// Mitsubishi GX Works2 project: PLC_GROUP_37   PLC: FX3G

// global labels: Global1
VAR_GLOBAL
  Day_Active_Light AT Y007 : BOOL;
  Emergency_Stop AT X005 : BOOL;
  Start_Day_Switch AT X007 : BOOL;
  Raspberry_Stock AT D1110 : REAL;
  Lemon_Stock AT D1120 : REAL;
  Stabilizer_Stock AT D1130 : REAL;
  Gummy_Stock AT D1140 : REAL;
  Total_Packages AT D1150 : REAL;
  Raspberry_Input AT D1160 : REAL;
  Lemon_Input AT D1170 : REAL;
  Stabilizer_Input AT D1180 : REAL;
  Gummy_Input AT D1190 : REAL;
END_VAR
VAR_GLOBAL CONSTANT
  Constant_0 : REAL;
END_VAR
VAR_GLOBAL
  End_Day_Flag AT M0 : BOOL;
  Start_Production_Switch AT X001 : BOOL;
  Analog_Input_1 AT D8280 : INT;
  Sampled_Package_Type AT D1100 : REAL;
  Regular_Selected AT M1 : BOOL;
  Luxury_Selected AT M3 : BOOL;
  Inventory_OK AT M5 : BOOL;
END_VAR
VAR_GLOBAL CONSTANT
  Constant_5 : REAL := 5;
  Constant_6 : REAL := 6;
  Constant_280 : REAL := 280;
  Constant_455 : REAL := 455;  (* ֶ *)
  Constant_105 : REAL := 105;
  Constant_385 : REAL := 385;
  Constant_28 : REAL := 28;
  Constant_665 : REAL := 665;
  Constant_210 : REAL := 210;
  Constant_70 : REAL := 70;
END_VAR
VAR_GLOBAL
  Luxury_Inv_OK AT M11 : BOOL;
  Regular_Inv_OK AT M9 : BOOL;
END_VAR
VAR_GLOBAL CONSTANT
  Constant_50_Int : INT := 50;
END_VAR
VAR_GLOBAL
  PrepT_Coil AT TC0 : BOOL;
  PrepT_Contact AT TS0 : BOOL;
  Ice_Cream_Prep_Light AT Y000 : BOOL;
END_VAR
VAR_GLOBAL CONSTANT
  Constant_1 : REAL := 1;
END_VAR
VAR_GLOBAL
  Analog_Output AT D8282 : INT;
  Wait_For_Cooling AT M13 : BOOL;
  Cooling_Active AT M15 : BOOL;
  Cooling_Light AT Y002 : BOOL;
  CoolingT_Coil AT TC1 : BOOL;
  CoolingT_Contact AT TS1 : BOOL;
  Start_Cooling_Switch AT X002 : BOOL;
  Temp_Sensor_10_Deg AT X003 : BOOL;
END_VAR
VAR_GLOBAL CONSTANT
  Constant_80_Int : INT := 80;
END_VAR
VAR_GLOBAL
  Mixing_Active AT M17 : BOOL;
  MixT_Reg_Coil AT TC2 : BOOL;
  MixT_Reg_Contact AT TS2 : BOOL;
  MixT_Lux_Coil AT TC3 : BOOL;
  MixT_Lux_Contact AT TS3 : BOOL;
  Mix_Light_1 AT Y005 : BOOL;
  Mix_Light_2 AT Y006 : BOOL;
END_VAR
VAR_GLOBAL CONSTANT
  Constant_30_Int : INT := 30;
END_VAR
VAR_GLOBAL
  BlinkT1_Coil AT TC4 : BOOL;
  BlinkT1_Contact AT TS4 : BOOL;
  BlinkT2_Coil AT TC5 : BOOL;
  BlinkT2_Contact AT TS5 : BOOL;
END_VAR
VAR_GLOBAL CONSTANT
  Constant_10_Int : INT := 10;
END_VAR
VAR_GLOBAL
  Process_Active AT M21 : BOOL;
  R_Reg_OK AT M23 : BOOL;
  L_Reg_OK AT M25 : BOOL;
  S_Reg_OK AT M27 : BOOL;
  G_Reg_OK AT M29 : BOOL;
  R_Lux_OK AT M31 : BOOL;
  L_Lux_OK AT M33 : BOOL;
  S_Lux_OK AT M35 : BOOL;
  G_Lux_OK AT M37 : BOOL;
  QC_Counter AT CC0 : BOOL;
END_VAR
VAR_GLOBAL CONSTANT
  Constant_15_Int : INT := 15;
END_VAR
VAR_GLOBAL
  QC_Timer AT TC10 : BOOL;
  QC_Sampling_Flag AT M50 : BOOL;
  Global_Low_Stock AT M52 : BOOL;
END_VAR
VAR_GLOBAL CONSTANT
  Constant_1000 : REAL := 1000;
END_VAR

// task Task_01 (event TRUE, interval 0, priority 31): POU_01

PROGRAM POU_01
(* structured ladder/FBD written out as ST: instructions are called as NAME(EN, inputs, outputs); _pN, _eN, _tN stand for wires *)
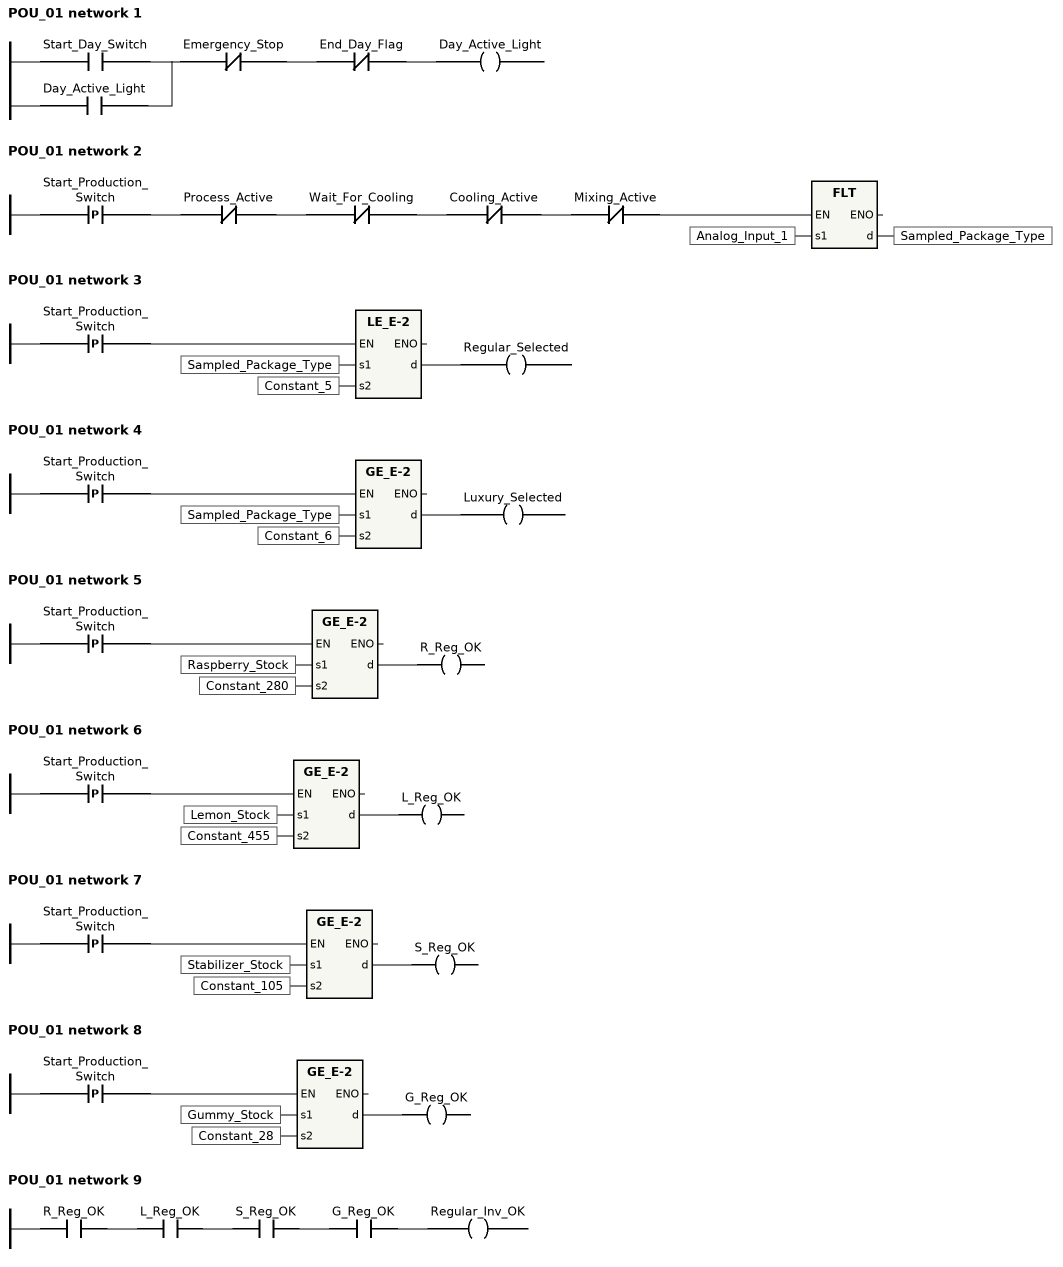
(* network 1 *)
Day_Active_Light := ((Start_Day_Switch OR Day_Active_Light) AND NOT Emergency_Stop) AND NOT End_Day_Flag;
(* network 2 *)
FLT(LDP(TRUE, Start_Production_Switch) AND NOT Process_Active AND NOT Wait_For_Cooling AND NOT Cooling_Active AND NOT Mixing_Active, Analog_Input_1, Sampled_Package_Type);
(* network 3 *)
LE_E(LDP(TRUE, Start_Production_Switch), Sampled_Package_Type, Constant_5, _t1);
Regular_Selected := _t1;
(* network 4 *)
GE_E(LDP(TRUE, Start_Production_Switch), Sampled_Package_Type, Constant_6, _t1);
Luxury_Selected := _t1;
(* network 5 *)
GE_E(LDP(TRUE, Start_Production_Switch), Raspberry_Stock, Constant_280, _t1);
R_Reg_OK := _t1;
(* network 6 *)
GE_E(LDP(TRUE, Start_Production_Switch), Lemon_Stock, Constant_455, _t1);
L_Reg_OK := _t1;
(* network 7 *)
GE_E(LDP(TRUE, Start_Production_Switch), Stabilizer_Stock, Constant_105, _t1);
S_Reg_OK := _t1;
(* network 8 *)
GE_E(LDP(TRUE, Start_Production_Switch), Gummy_Stock, Constant_28, _t1);
G_Reg_OK := _t1;
(* network 9 *)
Regular_Inv_OK := R_Reg_OK AND L_Reg_OK AND S_Reg_OK AND G_Reg_OK;
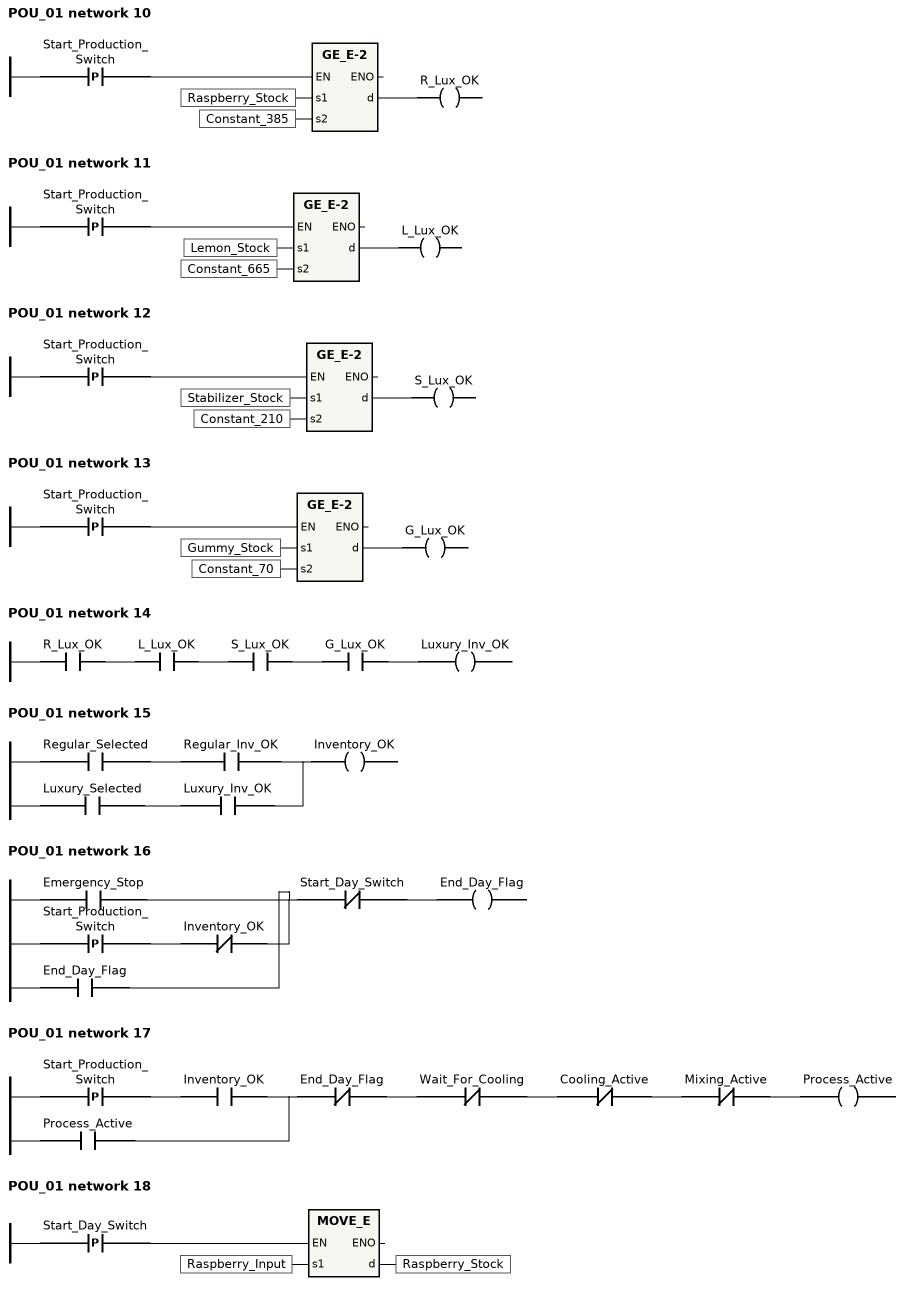
(* network 10 *)
GE_E(LDP(TRUE, Start_Production_Switch), Raspberry_Stock, Constant_385, _t1);
R_Lux_OK := _t1;
(* network 11 *)
GE_E(LDP(TRUE, Start_Production_Switch), Lemon_Stock, Constant_665, _t1);
L_Lux_OK := _t1;
(* network 12 *)
GE_E(LDP(TRUE, Start_Production_Switch), Stabilizer_Stock, Constant_210, _t1);
S_Lux_OK := _t1;
(* network 13 *)
GE_E(LDP(TRUE, Start_Production_Switch), Gummy_Stock, Constant_70, _t1);
G_Lux_OK := _t1;
(* network 14 *)
Luxury_Inv_OK := R_Lux_OK AND L_Lux_OK AND S_Lux_OK AND G_Lux_OK;
(* network 15 *)
Inventory_OK := (Regular_Selected AND Regular_Inv_OK) OR (Luxury_Selected AND Luxury_Inv_OK);
(* network 16 *)
End_Day_Flag := (Emergency_Stop OR (LDP(TRUE, Start_Production_Switch) AND NOT Inventory_OK) OR End_Day_Flag) AND NOT Start_Day_Switch;
(* network 17 *)
Process_Active := (((((LDP(TRUE, Start_Production_Switch) AND Inventory_OK) OR Process_Active) AND NOT End_Day_Flag) AND NOT Wait_For_Cooling) AND NOT Cooling_Active) AND NOT Mixing_Active;
(* network 18 *)
MOVE_E(LDP(TRUE, Start_Day_Switch), Raspberry_Input, Raspberry_Stock);
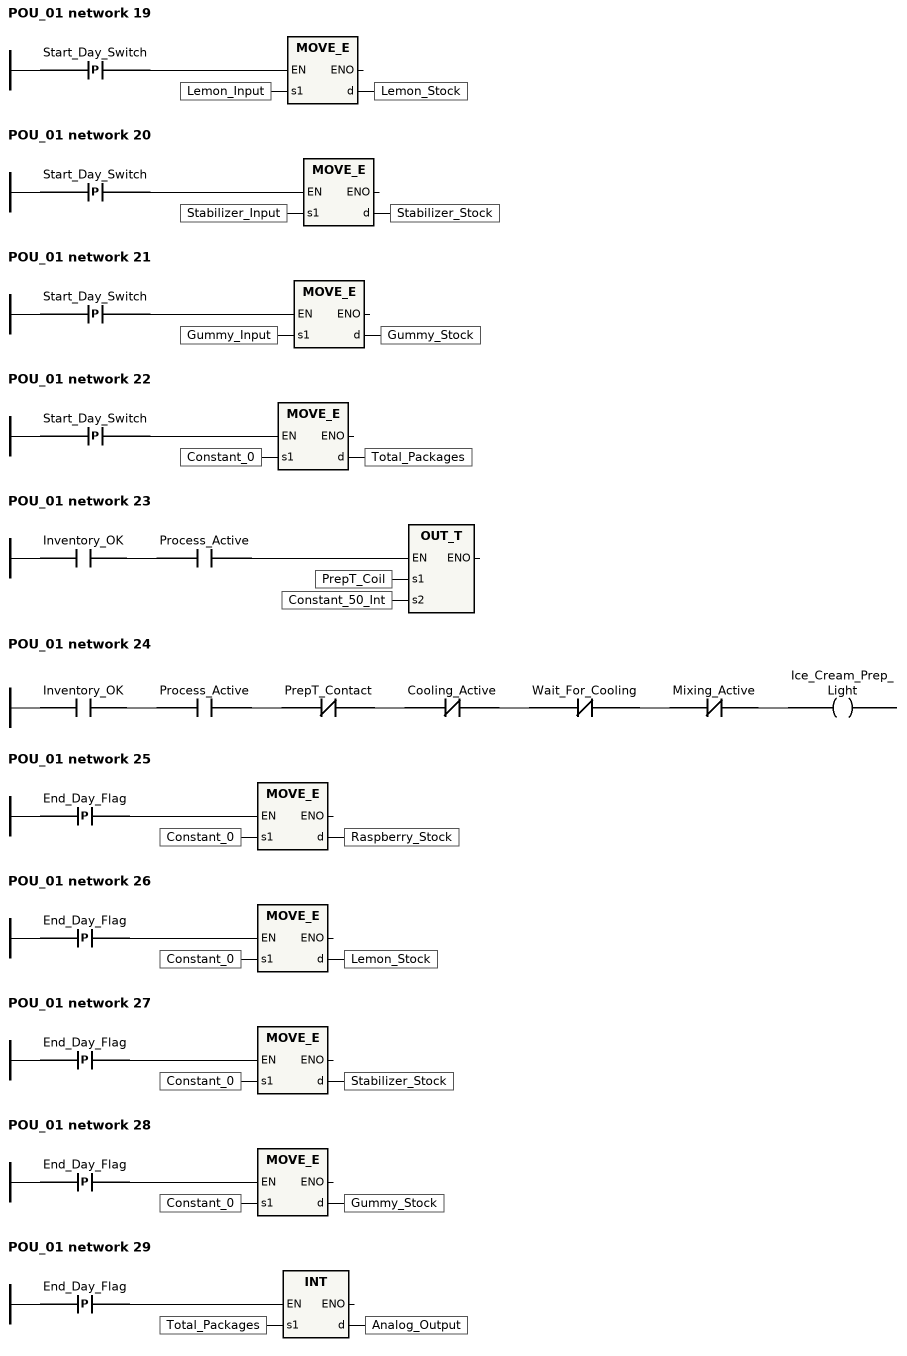
(* network 19 *)
MOVE_E(LDP(TRUE, Start_Day_Switch), Lemon_Input, Lemon_Stock);
(* network 20 *)
MOVE_E(LDP(TRUE, Start_Day_Switch), Stabilizer_Input, Stabilizer_Stock);
(* network 21 *)
MOVE_E(LDP(TRUE, Start_Day_Switch), Gummy_Input, Gummy_Stock);
(* network 22 *)
MOVE_E(LDP(TRUE, Start_Day_Switch), Constant_0, Total_Packages);
(* network 23 *)
OUT_T(Inventory_OK AND Process_Active, PrepT_Coil, Constant_50_Int);
(* network 24 *)
Ice_Cream_Prep_Light := Inventory_OK AND Process_Active AND NOT PrepT_Contact AND NOT Cooling_Active AND NOT Wait_For_Cooling AND NOT Mixing_Active;
(* network 25 *)
MOVE_E(LDP(TRUE, End_Day_Flag), Constant_0, Raspberry_Stock);
(* network 26 *)
MOVE_E(LDP(TRUE, End_Day_Flag), Constant_0, Lemon_Stock);
(* network 27 *)
MOVE_E(LDP(TRUE, End_Day_Flag), Constant_0, Stabilizer_Stock);
(* network 28 *)
MOVE_E(LDP(TRUE, End_Day_Flag), Constant_0, Gummy_Stock);
(* network 29 *)
INT(LDP(TRUE, End_Day_Flag), Total_Packages, Analog_Output);
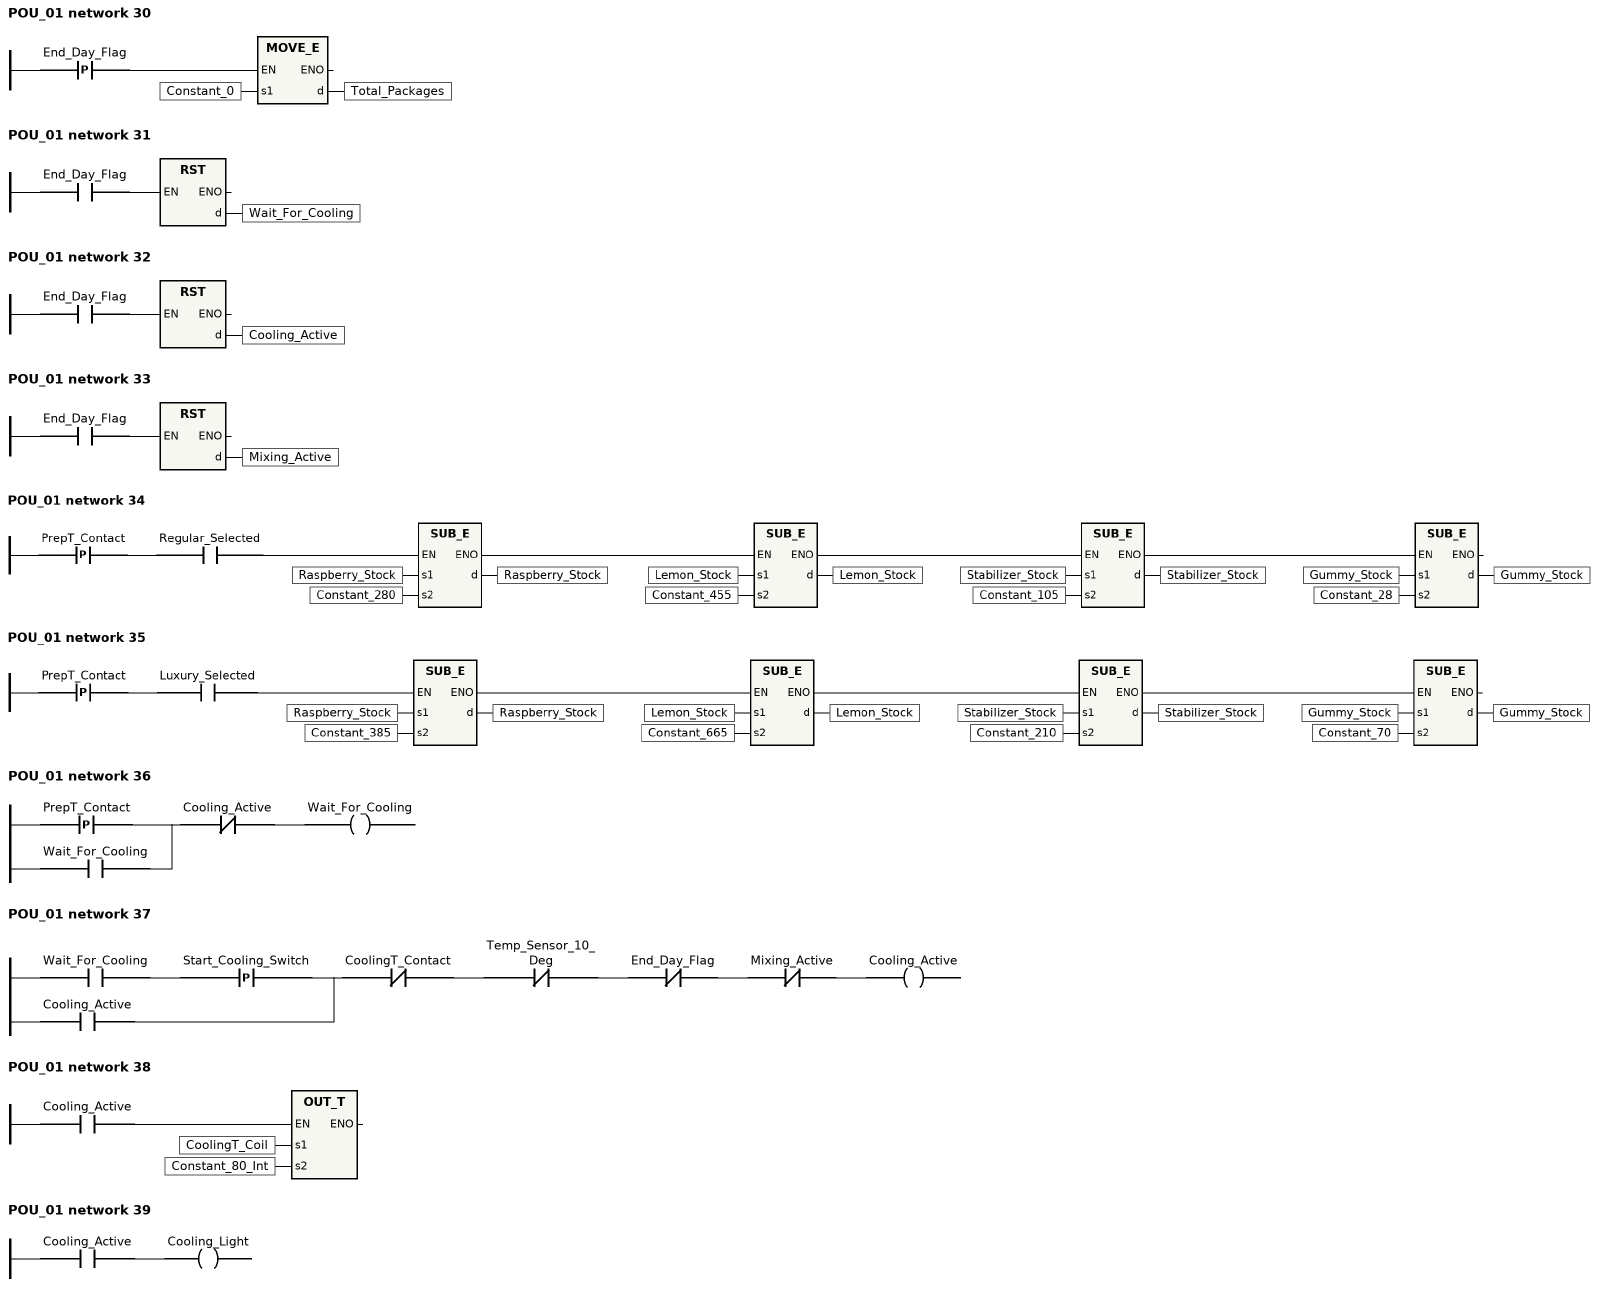
(* network 30 *)
MOVE_E(LDP(TRUE, End_Day_Flag), Constant_0, Total_Packages);
(* network 31 *)
RST(End_Day_Flag, Wait_For_Cooling);
(* network 32 *)
RST(End_Day_Flag, Cooling_Active);
(* network 33 *)
RST(End_Day_Flag, Mixing_Active);
(* network 34 *)
_e1 := SUB_E(LDP(TRUE, PrepT_Contact) AND Regular_Selected, Raspberry_Stock, Constant_280, Raspberry_Stock);
_e2 := SUB_E(_e1, Lemon_Stock, Constant_455, Lemon_Stock);
_e3 := SUB_E(_e2, Stabilizer_Stock, Constant_105, Stabilizer_Stock);
SUB_E(_e3, Gummy_Stock, Constant_28, Gummy_Stock);
(* network 35 *)
_e1 := SUB_E(LDP(TRUE, PrepT_Contact) AND Luxury_Selected, Raspberry_Stock, Constant_385, Raspberry_Stock);
_e2 := SUB_E(_e1, Lemon_Stock, Constant_665, Lemon_Stock);
_e3 := SUB_E(_e2, Stabilizer_Stock, Constant_210, Stabilizer_Stock);
SUB_E(_e3, Gummy_Stock, Constant_70, Gummy_Stock);
(* network 36 *)
Wait_For_Cooling := (LDP(TRUE, PrepT_Contact) OR Wait_For_Cooling) AND NOT Cooling_Active;
(* network 37 *)
Cooling_Active := (((((Wait_For_Cooling AND LDP(TRUE, Start_Cooling_Switch)) OR Cooling_Active) AND NOT CoolingT_Contact) AND NOT Temp_Sensor_10_Deg) AND NOT End_Day_Flag) AND NOT Mixing_Active;
(* network 38 *)
OUT_T(Cooling_Active, CoolingT_Coil, Constant_80_Int);
(* network 39 *)
Cooling_Light := Cooling_Active;
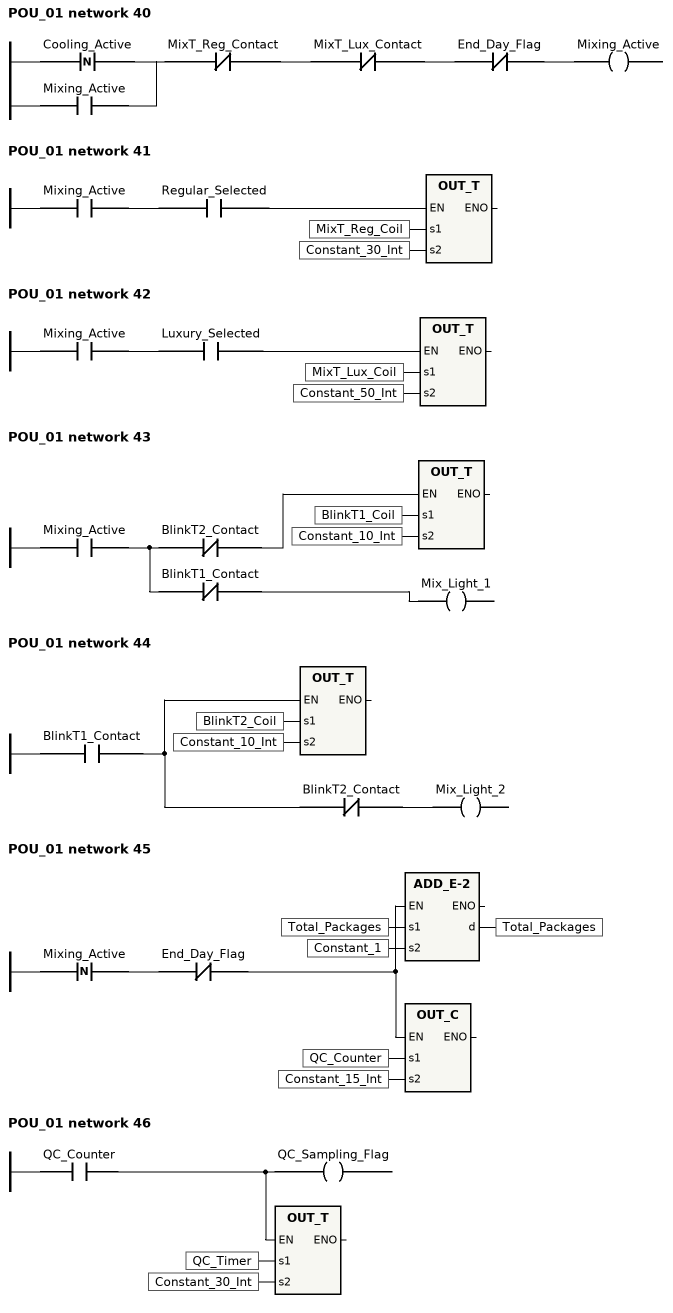
(* network 40 *)
Mixing_Active := (((LDF(TRUE, Cooling_Active) OR Mixing_Active) AND NOT MixT_Reg_Contact) AND NOT MixT_Lux_Contact) AND NOT End_Day_Flag;
(* network 41 *)
OUT_T(Mixing_Active AND Regular_Selected, MixT_Reg_Coil, Constant_30_Int);
(* network 42 *)
OUT_T(Mixing_Active AND Luxury_Selected, MixT_Lux_Coil, Constant_50_Int);
(* network 43 *)
OUT_T(Mixing_Active AND NOT BlinkT2_Contact, BlinkT1_Coil, Constant_10_Int);
Mix_Light_1 := Mixing_Active AND NOT BlinkT1_Contact;
(* network 44 *)
OUT_T(BlinkT1_Contact, BlinkT2_Coil, Constant_10_Int);
Mix_Light_2 := BlinkT1_Contact AND NOT BlinkT2_Contact;
(* network 45 *)
_p1 := LDF(TRUE, Mixing_Active) AND NOT End_Day_Flag;
ADD_E(_p1, Total_Packages, Constant_1, Total_Packages);
OUT_C(_p1, QC_Counter, Constant_15_Int);
(* network 46 *)
QC_Sampling_Flag := QC_Counter;
OUT_T(QC_Counter, QC_Timer, Constant_30_Int);
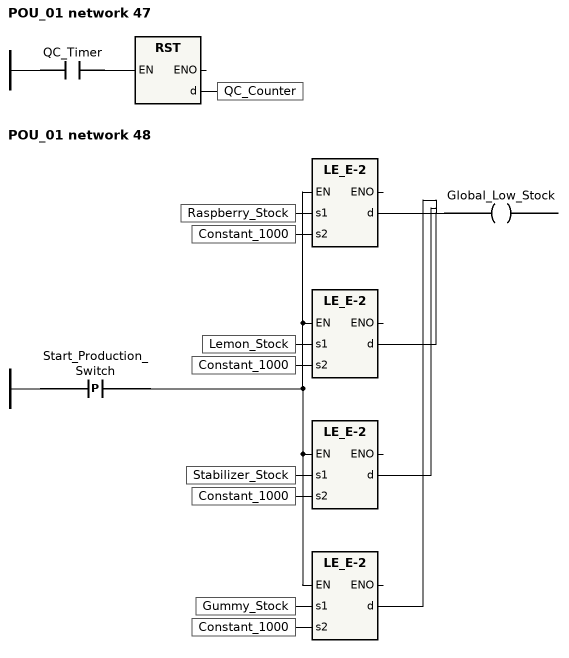
(* network 47 *)
RST(QC_Timer, QC_Counter);
(* network 48 *)
_p1 := LDP(TRUE, Start_Production_Switch);
LE_E(_p1, Raspberry_Stock, Constant_1000, _t2);
LE_E(_p1, Lemon_Stock, Constant_1000, _t3);
LE_E(_p1, Stabilizer_Stock, Constant_1000, _t4);
LE_E(_p1, Gummy_Stock, Constant_1000, _t5);
Global_Low_Stock := _t2 OR _t3 OR _t4 OR _t5;
END_PROGRAM
